FUNCTION_BLOCK AUTOMATIC_SCREW_PICKUP_TEST
VAR_INPUT
END_VAR
VAR_OUTPUT
END_VAR
VAR
END_VAR

ACTION ACT_SEQUENCE_CHAIN:
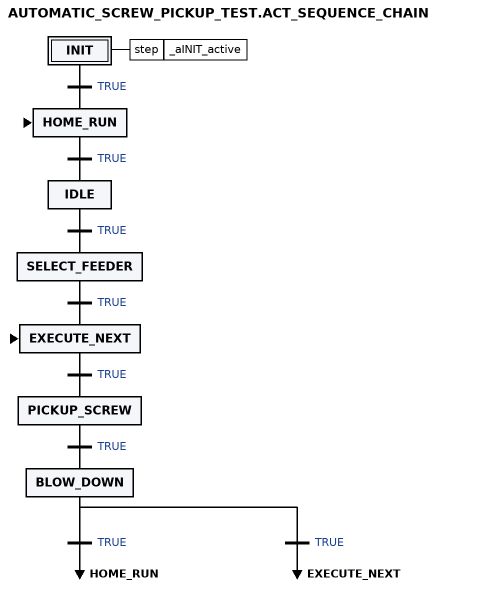
INITIAL_STEP INIT:
    _aINIT_active(N);  // step action
END_STEP
TRANSITION FROM INIT TO HOME_RUN
    := TRUE;
END_TRANSITION
STEP HOME_RUN:
END_STEP
TRANSITION FROM HOME_RUN TO IDLE
    := TRUE;
END_TRANSITION
STEP IDLE:
END_STEP
TRANSITION FROM IDLE TO SELECT_FEEDER
    := TRUE;
END_TRANSITION
STEP SELECT_FEEDER:
END_STEP
TRANSITION FROM SELECT_FEEDER TO EXECUTE_NEXT
    := TRUE;
END_TRANSITION
STEP EXECUTE_NEXT:
END_STEP
TRANSITION FROM EXECUTE_NEXT TO PICKUP_SCREW
    := TRUE;
END_TRANSITION
STEP PICKUP_SCREW:
END_STEP
TRANSITION FROM PICKUP_SCREW TO BLOW_DOWN
    := TRUE;
END_TRANSITION
STEP BLOW_DOWN:
END_STEP
TRANSITION FROM BLOW_DOWN TO HOME_RUN
    := TRUE;
END_TRANSITION
TRANSITION FROM BLOW_DOWN TO EXECUTE_NEXT
    := TRUE;
END_TRANSITION
// branch label Branch0_ACT_SEQUENCE_CHAIN
END_ACTION

END_FUNCTION_BLOCK

(* stored: Version 1.1.0.1, ProductVersion 3.1.4022.18
   POU AUTOMATIC_SCREW_PICKUP_TEST: Id {4cb08561-5be3-47cc-b299-483650213744}, SpecialFunc None
   Action ACT_SEQUENCE_CHAIN: Id {15c146b8-8bc8-4b01-a5d3-a7fe0d9aaf88} *)
